TYPE ST_OerlikonPTM EXTENDS ST_PTM :
STRUCT
(* Extension of the PTM archetype for Oerlikon turbo controllers 
Applicable to: 
Mag Drive Digital
Mag Drive S
More?
*)
//Readbacks
	i_xDecel	:	BOOL;
	i_diPumpTemp:	DINT;
	i_diPwr   :   DINT;
	i_diElecTemp: DINT;

//Controls
	q_xRemote : BOOL; (* Remote control enabled *)

END_STRUCT
END_TYPE

(* stored: Version 1.1.0.1, ProductVersion 3.1.4018.5
   DUT ST_OerlikonPTM: Id {928359f7-41f5-4b97-ac89-aed21155294b} *)
